// TIA Portal V20 export
DATA_BLOCK "SBK08"   // DB321
// stored: MemoryReserve 100
   VAR
      "SAFETY DOOR LOCK1.INPUT" : Bool := TRUE;
      "SAFETY DOOR LOCK2.INPUT" : Bool := TRUE;
      "SAFETY DOOR LOCK3.INPUT" : Bool := TRUE;
      SPARE : Bool := FALSE;
      "SAFETY DOOR LOCK1.INPUT_1" : Bool := FALSE;
      "SAFETY DOOR LOCK2.INPUT_1" : Bool := FALSE;
      "SAFETY DOOR LOCK3.INPUT_1" : Bool := FALSE;
      SPARE_1 : Bool := FALSE;
      "SAFETY DOOR LOCK1.OUTPUT" : Bool := FALSE;
      "SAFETY DOOR LOCK2.OUTPUT" : Bool := FALSE;
      "SAFETY DOOR LOCK3.OUTPUT" : Bool := FALSE;
   END_VAR
BEGIN
END_DATA_BLOCK
